TYPE DUT :
STRUCT
END_STRUCT
END_TYPE

(* stored: Version 1.1.0.1, ProductVersion 3.1.4024.10
   DUT DUT: Id {4430ce7c-ea99-478c-b9d5-9777e40a169a} *)
